FUNCTION_BLOCK Stamp_StampWorkpiece EXTENDS ControlPrimitiveBase
VAR_INPUT
END_VAR
VAR_OUTPUT
END_VAR
VAR
	// (EProcessVariables.Stamp_WorkpieceState = 1) AND (EProcessVariables.Stamp_WPAtStamp = TRUE)
	m_compExpr273: ComparisonExpression(EProcessVariables.Stamp_WorkpieceState, EComparisonType.equals, EDataType.numeric, FALSE, 1, '', TRUE);
	m_compExpr275: ComparisonExpression(EProcessVariables.Stamp_WPAtStamp, EComparisonType.equals, EDataType.binary, TRUE, 0, '', TRUE);
	m_precondition: BoolExpression(m_compExpr273, EBoolOperation.and_op, m_compExpr275);
	
	// EProcessVariables.Stamp_WorkpieceState = 2
	m_postcondition: ComparisonExpression(EProcessVariables.Stamp_WorkpieceState, EComparisonType.equals, EDataType.numeric, FALSE, 2, '', TRUE);

	m_ptrStamp: POINTER TO Stamp;
	
	m_step: INT := 0;
	t_Stamp : TON;
END_VAR

SUPER^();

METHOD Abort : BOOL
VAR_INPUT
END_VAR
m_ptrStamp^.m_stampingCylinder.METH_Retract();
m_ptrStamp^.m_slidingCylinder.METH_Extend();
Abort := TRUE;
END_METHOD

(* Execution logic of this Control Primitive. *)
METHOD PROTECTED ExecuteInternal : BOOL
VAR_INPUT
	(*
	 * pressure_white: INT
	 * pressure_black: INT
	 * pressure_metal: INT
	 *)
	i_params: ParameterSet;
END_VAR
VAR
	m_pressureVal: SValue;
END_VAR
ExecuteInternal := FALSE;

CASE m_step OF
	0: // take in wp
	m_ptrStamp^.m_slidingCylinder.METH_Retract();
	IF m_ptrStamp^.m_slidingCylinder.Retracted THEN
		m_step := 1;
	END_IF
	
	1: // stamp wp
	m_ptrStamp^.StampPressure := GetPressure(i_params);
	m_ptrStamp^.m_stampingCylinder.METH_Extend();
	t_Stamp(IN:=TRUE, PT:=T#1500MS);
	IF t_Stamp.Q THEN
		IF m_ptrStamp^.StampPressure >= m_pressureVal.Value.Numeric THEN
			m_step := 2;
			t_Stamp(IN:=FALSE);
		END_IF
	END_IF
	
	2: // retract stamp
	m_ptrStamp^.m_stampingCylinder.METH_Retract();
	IF m_ptrStamp^.m_stampingCylinder.Retracted THEN
		m_step := 3;
	END_IF
	
	3: // provide wp
	m_ptrStamp^.m_slidingCylinder.METH_Extend();
	IF m_ptrStamp^.m_slidingCylinder.Extended THEN
		m_step := 0;
		ExecuteInternal := TRUE;
	END_IF
END_CASE
END_METHOD

METHOD FB_init : BOOL
VAR_INPUT
	bInitRetains : BOOL; // if TRUE, the retain variables are initialized (warm start / cold start)
	bInCopyCode : BOOL;  // if TRUE, the instance afterwards gets moved into the copy code (online change)
	
	i_ptrStamp: POINTER TO Stamp;
END_VAR
m_ptrStamp := i_ptrStamp;

m_id := EPrimitives.Stamp_StampWorkpiece;
m_timeout := T#200S;
m_paramDefinition := 'pressure_white:INT;pressure_black:INT;pressure_metal:INT;';

Precondition := m_precondition;
Postcondition := m_postcondition;
END_METHOD

METHOD PRIVATE GetPressure : INT
VAR_INPUT
	(*
	 * pressure_white: INT
	 * pressure_black: INT
	 * pressure_metal: INT
	 *)
	i_params: ParameterSet;
END_VAR
VAR
	m_pressureVal: SValue;
END_VAR
CASE LREAL_TO_UINT(m_st^.GetNumeric(EProcessVariables.Stamp_ProductType)) OF
	EProductTypes.white:
		m_pressureVal := i_params.Retrieve('pressure_white');
		GetPressure := LREAL_TO_INT(m_pressureVal.Value.Numeric);
	EProductTypes.black:
		m_pressureVal := i_params.Retrieve('pressure_black');
		GetPressure := LREAL_TO_INT(m_pressureVal.Value.Numeric);
	EProductTypes.metal:
		m_pressureVal := i_params.Retrieve('pressure_metal');
		GetPressure := LREAL_TO_INT(m_pressureVal.Value.Numeric);
	ELSE
		GetPressure := 0;
END_CASE
END_METHOD

END_FUNCTION_BLOCK

(* stored: Version 1.1.0.1, ProductVersion 3.1.4024.12
   POU Stamp_StampWorkpiece: Id {43a8f1ee-c4bc-4d50-abf6-1a0e6209c669}, SpecialFunc None
   Method Abort: Id {4b258602-9728-45da-88a5-82994e93e50a}
   Method ExecuteInternal: Id {20ea73f5-52e1-4027-b77b-4b90b04c41c4}
   Method FB_init: Id {ae19cc40-2395-457d-a4db-026b5c45012b}
   Method GetPressure: Id {a758e95a-746f-4659-933f-dd77eb48177a} *)
